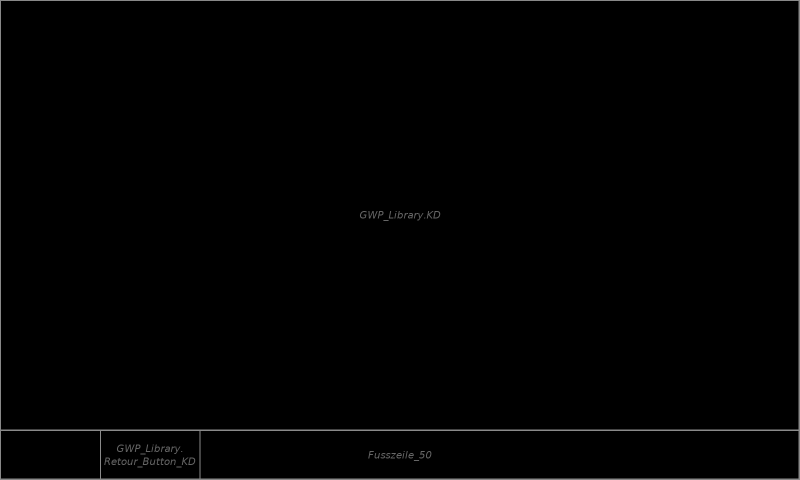
VISUALIZATION KD  // 800x480
    Frame (0,0 800x430)
        shows GWP_Library.KD(FB_KD := Main.KD_0)
    Group (0,430 800x50)
        Frame (0,0 800x50)
            shows Fusszeile_50()
        Frame (100,0 100x50)
            shows GWP_Library.Retour_Button_KD()
END_VISUALIZATION

(* stored: Version 1.1.0.1, ProductVersion 3.1.4022.6
   Visu KD: Id {b57b8b82-dee3-4459-8fe9-80811bf92d0e} *)
